// TwinCAT 3 PLC project separator
// ProgramVersion: 3.1.4023.0
// libraries:
//   Tc2_DataExchange, * (Beckhoff Automation GmbH)
//   Tc2_Standard, * (Beckhoff Automation GmbH)
//   Tc2_System, * (Beckhoff Automation GmbH)
//   Tc3_Module, * (Beckhoff Automation GmbH)
// project tree:
//   FB/ FB_ReadAmsValue.TcPOU (not stored), FB_WriteAmsValue.TcPOU (not stored)
//   GVLs/ GVL.TcGVL, SUPVams.TcGVL (not stored)
//   / PlcTask.TcTTO
//   POUs/ MAIN.TcPOU, POU_readSupvData.TcPOU, POU_writeSeparatorToSupvData.TcPOU
// real-time tasks:
//   TASK PlcTask: cycle T#10ms, priority 20, ADS port 350

CONFIGURATION separator
    RESOURCE PLC ON TwinCAT3
        TASK PlcTask(INTERVAL := T#10ms, PRIORITY := 20);
        PROGRAM MAIN WITH PlcTask : MAIN;
    END_RESOURCE
END_CONFIGURATION

// ---- GVLs/GVL.TcGVL
{attribute 'qualified_only'}
VAR_GLOBAL
	// setpoints
	PROD_RATE_SP					:	LREAL	:= 22.89;	// production rate
	L_STRIPPER_SP					:	LREAL	:= 50.0;	// stripper level
	L_SEPARATOR_SP					:	LREAL	:= 50.0;	// separator level
	L_REACTOR_SP					:	LREAL	:= 65.0;	// reactor level
	P_REACTOR_SP					:	LREAL;	// reactor pressure
	PCT_G_SP						:	LREAL;	// Mole percent G
	YA_SP							: 	LREAL;	// yA 
	YAC_SP							:	LREAL;	// yAC
	T_REACTOR_SP					:	LREAL;	// reactor temperature
	RECYC_VALVE_SP					:	LREAL;	// Recycle valve position
	STEAM_VALVE_SP					:	LREAL;	// Steam valve position
	L_AGITATOR_SP					:	LREAL;	// agitator setting		
	
	// Intermediate values
	Fp							:	LREAL; 		

	// actual production metrics
	COST						:	LREAL :=0.0;
	PctG						:	LREAL :=0.0;

	// process variables
	XMEAS						:	ARRAY[1..41] OF LREAL;
	XMEAS_TO_SUPV				:	ARRAY[1..16] OF LREAL; // 10,11-14,20,22,29-36
	
	XMV							:	ARRAY[1..12] OF LREAL;
	XMV_TO_SUPV					:	ARRAY[1..3] OF LREAL;  // 5,6,7
	
	// intermediate variables
	SEP_TEMP_SP					:	LREAL;	// separator temperaure setpoint
	RI							:	ARRAY[1..6] OF LREAL;	// ratio trimming outputs
	EADJ						:	LREAL;	// adjustment to production rate
	PCTG_SP						:	LREAL;	// setpoint for precent G
	
	// shutdown indicator
	SD_FLAG						: 	BOOL	:= FALSE;

	// operating time
	OPTIME					:	LREAL := 0.0;		
END_VAR

// ---- POUs/MAIN.TcPOU
PROGRAM MAIN
VAR
END_VAR

POU_readSupvData();
POU_writeSeparatorToSupvData();

END_PROGRAM

// ---- POUs/POU_readSupvData.TcPOU
PROGRAM POU_readSupvData
VAR
	sNetId: T_AmsNetId := SUPVams.sNetId;	// '5.30.23.91.1.1';
	nPort: T_AmsPort := SUPVams.nPort; 		// 851
	
	FB_ReadAmsValue_Fp: FB_ReadAmsValue;
	FB_ReadAmsValue_SepLevel: FB_ReadAmsValue;
	FB_ReadAmsValue_R5: FB_ReadAmsValue;
	nFpReadErrorId: UDINT;
	bFpReadError: BOOL;
	nSepLevelReadErrorId: UDINT;
	nR5ReadErrorId: UDINT;
	bSepLevelReadError: BOOL;
	bR5ReadError: BOOL;
END_VAR

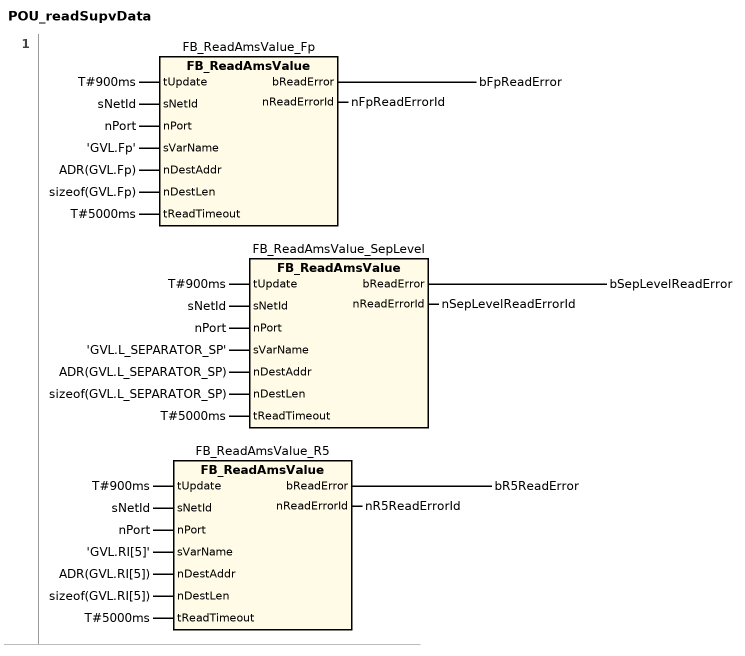
// NETWORK 1
FB_ReadAmsValue_Fp(
    tUpdate := T#900ms,
    sNetId := sNetId,
    nPort := nPort,
    sVarName := 'GVL.Fp',
    nDestAddr := ADR(GVL.Fp),
    nDestLen := sizeof(GVL.Fp),
    tReadTimeout := T#5000ms,
    nReadErrorId => nFpReadErrorId); // FB_ReadAmsValue
bFpReadError := FB_ReadAmsValue_Fp.bReadError;
FB_ReadAmsValue_SepLevel(
    tUpdate := T#900ms,
    sNetId := sNetId,
    nPort := nPort,
    sVarName := 'GVL.L_SEPARATOR_SP',
    nDestAddr := ADR(GVL.L_SEPARATOR_SP),
    nDestLen := sizeof(GVL.L_SEPARATOR_SP),
    tReadTimeout := T#5000ms,
    nReadErrorId => nSepLevelReadErrorId); // FB_ReadAmsValue
bSepLevelReadError := FB_ReadAmsValue_SepLevel.bReadError;
FB_ReadAmsValue_R5(
    tUpdate := T#900ms,
    sNetId := sNetId,
    nPort := nPort,
    sVarName := 'GVL.RI[5]',
    nDestAddr := ADR(GVL.RI[5]),
    nDestLen := sizeof(GVL.RI[5]),
    tReadTimeout := T#5000ms,
    nReadErrorId => nR5ReadErrorId); // FB_ReadAmsValue
bR5ReadError := FB_ReadAmsValue_R5.bReadError;

END_PROGRAM

// ---- POUs/POU_writeSeparatorToSupvData.TcPOU
PROGRAM POU_writeSeparatorToSupvData
VAR
	sNetId: T_AmsNetId := SUPVams.sNetId;	// '5.30.23.91.1.1';
	nPort: T_AmsPort := SUPVams.nPort; 		// 851	

	FB_WriteAmsValue_XMEAS: FB_WriteAmsValue;
	FB_WriteAmsValue_XMV: FB_WriteAmsValue;
	nXMEASWriteErrorId: UDINT;
	bXMEASWriteError: BOOL;
	bXMVWriteError: BOOL;
	nXMVWriteErrorId: UDINT;
END_VAR

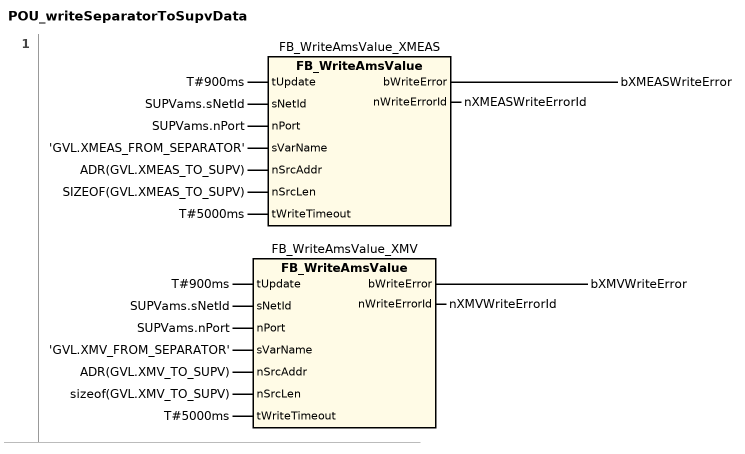
// NETWORK 1
FB_WriteAmsValue_XMEAS(
    tUpdate := T#900ms,
    sNetId := SUPVams.sNetId,
    nPort := SUPVams.nPort,
    sVarName := 'GVL.XMEAS_FROM_SEPARATOR',
    nSrcAddr := ADR(GVL.XMEAS_TO_SUPV),
    nSrcLen := SIZEOF(GVL.XMEAS_TO_SUPV),
    tWriteTimeout := T#5000ms,
    nWriteErrorId => nXMEASWriteErrorId); // FB_WriteAmsValue
bXMEASWriteError := FB_WriteAmsValue_XMEAS.bWriteError;
FB_WriteAmsValue_XMV(
    tUpdate := T#900ms,
    sNetId := SUPVams.sNetId,
    nPort := SUPVams.nPort,
    sVarName := 'GVL.XMV_FROM_SEPARATOR',
    nSrcAddr := ADR(GVL.XMV_TO_SUPV),
    nSrcLen := sizeof(GVL.XMV_TO_SUPV),
    tWriteTimeout := T#5000ms,
    nWriteErrorId => nXMVWriteErrorId); // FB_WriteAmsValue
bXMVWriteError := FB_WriteAmsValue_XMV.bWriteError;

END_PROGRAM
